FUNCTION_BLOCK FB_AO (* Service Interface Function Block Type *)
  (* Standard: 61499-2 *)
  (* Version 0.0, 2014-5-4, wildai, nxtControl GmbH, template *)
  (* Compiler Cpp nxtControl builtin 1.0 *)
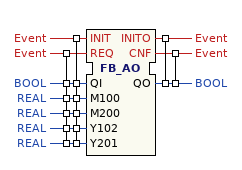
  EVENT_INPUT
    INIT WITH QI, M100, M200, Y102, Y201; (* Service Initialization *)
    REQ WITH QI, M100, M200, Y102, Y201; (* Service Request *)
  END_EVENT
  EVENT_OUTPUT
    INITO WITH QO; (* Initialization Confirm *)
    CNF WITH QO; (* Confirmation of Requested Service *)
  END_EVENT
  VAR_INPUT
    QI : BOOL; (* Event Input Qualifier *)
    M100 : REAL;
    M200 : REAL;
    Y102 : REAL;
    Y201 : REAL;
  END_VAR
  VAR_OUTPUT
    QO : BOOL; (* Event Output Qualifier *)
  END_VAR
  SERVICE FB_AO/RESOURCE
    SEQUENCE normal_establishment
      FB_AO.INIT+(PARAMS) -> RESOURCE.initialize(PARAMS) -> FB_AO.INITO+();
    END_SEQUENCE
    SEQUENCE unsuccessful_establishment
      FB_AO.INIT+(PARAMS) -> RESOURCE.initialize(PARAMS) -> FB_AO.INITO-(STATUS);
    END_SEQUENCE
    SEQUENCE request_confirm
      FB_AO.REQ+(SD) -> RESOURCE.request(SD) -> FB_AO.CNF+(RD);
    END_SEQUENCE
    SEQUENCE request_inhibited
      FB_AO.REQ-(SD) -> FB_AO.CNF-(STATUS);
    END_SEQUENCE
    SEQUENCE request_error
      FB_AO.REQ+(SD) -> RESOURCE.request(SD) -> FB_AO.CNF-(STATUS);
    END_SEQUENCE
    SEQUENCE indication_response
      FB_AO.RSP(QI,SD) -> RESOURCE.response(QI,SD);
      RESOURCE.indicate(RD) -> FB_AO.IND+(RD);
    END_SEQUENCE
    SEQUENCE indication_inhibited
      RESOURCE.indicate(RD,QI=FALSE) -> RESOURCE.inhibited();
    END_SEQUENCE
    SEQUENCE error_indication
      RESOURCE.error(STATUS) -> FB_AO.IND-(STATUS);
    END_SEQUENCE
    SEQUENCE application_initiated_termination
      FB_AO.INIT-() -> RESOURCE.terminate() -> FB_AO.INITO-(STATUS);
    END_SEQUENCE
    SEQUENCE resource_initiated_termination
      -> FB_AO.INITO-(STATUS);
    END_SEQUENCE
  END_SERVICE
END_FUNCTION_BLOCK
